FUNCTION_BLOCK DriverSequence
VAR_IN_OUT
	enable : BOOL;
	contUp : BOOL;
	contDown : BOOL;
	target : REAL;
END_VAR
VAR_OUTPUT
	ready : BOOL;
	
	busy : BOOL;
	position : REAL;
END_VAR
VAR
	driverSlider : ClearLinkEIP;
	
	step : INT;
	timer : TON;
END_VAR

driverSlider();

IF NOT driverSlider.homeSet THEN
	driverSlider.homingSequence();
	RETURN;
END_IF

driverSlider.bEnable := enable; //only confirm enable after home is set

driverSlider.stop();
IF contUp THEN
	driverSlider.moveContinuous(direction := MC_Positive_Direction);
	contDown := FALSE;
END_IF

IF contDown THEN
	driverSlider.moveContinuous(direction := MC_Negative_Direction);
	contUp := FALSE;
END_IF


IF target >= 0 THEN
	driverSlider.moveAbsolute(newTarget := target);
	//target := 0;
END_IF


IF driverSlider.innerLimit THEN
	contDown := FALSE;
END_IF
IF driverSlider.home THEN
	contUp := FALSE;
END_IF

position := driverSlider.position;
busy := driverSlider.busy;

METHOD autoSequence : BOOL
VAR_INPUT
END_VAR
timer(IN:= , PT:= , Q=> , ET=> );

CASE step OF
	0: //+continuous for 5s
		timer.IN := TRUE;
		timer.PT := T#5S;
		
		contUp := TRUE;
		
		IF timer.Q THEN
			timer.IN := FALSE;
			contUp := FALSE;
			step := 10;
		END_IF
		
	10: //target
		IF position = 150 AND NOT busy THEN
			target := -1;
			step := 20;
			RETURN;
		END_IF
		
		target := 150;
		
		IF busy THEN
			//step := 11;
		END_IF
		
	11:
		//paste top part of 10 if does not work
	
	20: //-continuous 2s
		timer.IN := TRUE;
		timer.PT := T#2S;
		
		contDown := TRUE;
		
		IF timer.Q THEN
			timer.IN := FALSE;
			contDown := FALSE;
			step := 30;
		END_IF
	
	
	30: //target 0
		target := 0;
		
		IF busy THEN
			step := 31;
		END_IF
		
	31:
		IF position = 0 AND NOT busy THEN
			target := -1;
			step := 40;
			RETURN;
		END_IF
		
	40:
		timer.IN := TRUE;
		timer.PT := T#1S;
		
		IF timer.Q THEN
			timer.IN := FALSE;
			step := 0;
		END_IF
END_CASE
END_METHOD

END_FUNCTION_BLOCK

(* stored: Version 1.1.0.1, ProductVersion 3.1.4024.11
   POU DriverSequence: Id {a3f9ba0a-2ad0-41b4-9a6e-1a63d7120b1c}, SpecialFunc None
   Method autoSequence: Id {ca498a70-55ce-48ed-a3ae-c5c08cfeb800} *)
